DATA_BLOCK "dbMain"
{ S7_Optimized_Access := 'TRUE' }
VERSION : 0.1
NON_RETAIN
"fbMain"

BEGIN
   Room[1].Rack[1].Fertigation.ShelvesFertigation[1].Controls.Flood_Duration := 1;
   Room[1].Rack[2].Fertigation.AI_Reservoir_Level.rHighCalibration := 100.0;
   Room[1].Rack[3].Fertigation.AI_Reservoir_Level.rHighCalibration := 0.0;

END_DATA_BLOCK

